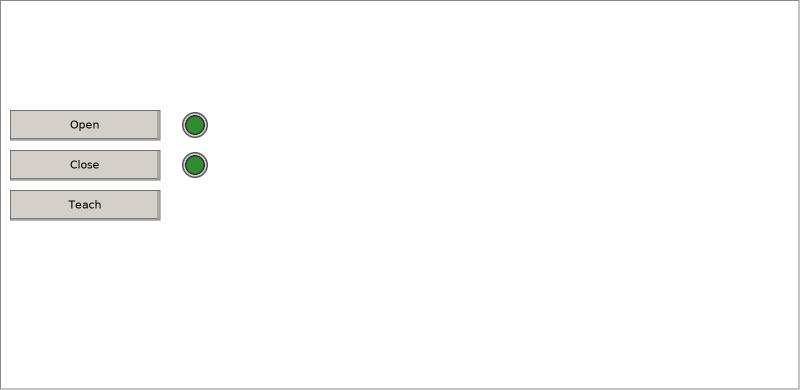
VISUALIZATION VisuValveControl  // 800x390
VAR_IN_OUT
	fbManualControler	: FB_ManualController ;
END_VAR
    Button (10,110 150x30), "Open"
        tap fbManualControler.pDevValve^.stManualCtrl.bCmdOpen
    Button (10,150 150x30), "Close"
        tap fbManualControler.pDevValve^.stManualCtrl.bCmdClose
    Lamp1 (180,110 30x30), variable: fbManualControler.pDevValve^.bFco_Open, style: Lamp-Lamp1-Green
    Button (10,190 150x30), "Teach"
        toggle fbManualControler.pDevValve^.stManualCtrl.bCmdTeach
    Lamp1 (180,150 30x30), variable: fbManualControler.pDevValve^.bFco_Closed, style: Lamp-Lamp1-Green
END_VISUALIZATION

(* stored: Version 1.1.0.1, ProductVersion 3.1.4024.9
   Visu VisuValveControl: Id {5822c885-21b0-4bb6-89f5-b6fde4df3f46} *)
